FUNCTION_BLOCK FB_Simulation
VAR_INPUT
	
END_VAR
VAR_OUTPUT

END_VAR
VAR
	//timers
	timTimerValueLong : TIME := T#7S;
	xTimerLongRunning: BOOL;

	timTimerValueShort : TIME := T#2S;
	xTimerShortRunning: BOOL;
	xTimerhmiRunning: BOOL;
	timTimerValuehmi: TIME := T#20MS;
END_VAR

//timer long and short for simulating wait time before somnething happens in the code
GVL.Timerlong(IN:=xTimerLongRunning, PT:=timTimerValueLong);
IF GVL.Timerlong.Q THEN
	xTimerLongRunning:=FALSE;
ELSE
	xTimerLongRunning:=TRUE;
END_IF

GVL.TimerShort(IN:=xTimerShortRunning, PT:=timTimerValueShort);
IF GVL.TimerShort.Q THEN
	xTimerShortRunning:=FALSE;
ELSE
	xTimerShortRunning:=TRUE;
END_IF

GVL.Timerhmi(IN:=xTimerhmiRunning, PT:=timTimerValuehmi);
IF GVL.Timerhmi.Q THEN
	xTimerhmiRunning:=FALSE;
ELSE
	xTimerhmiRunning:=TRUE;
END_IF

METHOD deplelitizerzuiger
VAR_INPUT
END_VAR
//als ciliderwerkt
IF i_xCilinderdepalitizerwerkt THEN
	//cilinder to wishsed positon
	main.fbDepalletizer.fbzuiger.eWistedHorizotalPosition;
END_IF

IF i_xHorizontalmovementWorking THEN
	//logica
END_IF
//als horizontaal werkt



// main.fbDepalletizer.fbZuiger.i_xEndSwitchIn := TRUE;
// main.fbDepalletizer.fbZuiger.i_xEndSwitchOut := TRUE;
// main.fbDepalletizer.fbZuiger.i_xHallSensorIn := TRUE;
// main.fbDepalletizer.fbZuiger.i_xHallSensorOut := TRUE;
// main.fbDepalletizer.fbZuiger.i_rPressureSensor := 4000;
END_METHOD

METHOD InvoerBuffer1
VAR_INPUT
END_VAR
//simulatie voor invoer buffer1

//klep

//sensor
END_METHOD

END_FUNCTION_BLOCK

(* stored: Version 1.1.0.1
   POU FB_Simulation: Id {9da5429a-6b68-472c-b1d4-54a90dc55476}, SpecialFunc None
   Method deplelitizerzuiger: Id {8051e9b7-c22e-4778-aa38-5be337bf3f0e}
   Method InvoerBuffer1: Id {2d9eb01e-8bfe-4d6d-bd0b-e4acfc4bf527} *)
